(* Logix 5000 project; controller FRC_CC_2020 vendor 1 type 14 code 150 rev 31.11; software revision 31.01; part 4 of 4 *)
(* tags used below, declared in another part *)
   Conn_Open : BOOL[32];
   Next_Write : BOOL[32];
   ONS : BOOL[64];
   ONS_B : BOOL[32];
   ONS_ERR : BOOL[32];
   RW_Instance : INT[20];
   RW_Select : DINT;
   MBTI_Read_Data_MSG_07 : MESSAGE;
   MBTI_Read_Data_MSG_08 : MESSAGE;
   MBTI_Read_Data_MSG_09 : MESSAGE;
   MBTI_Read_Done : BOOL[32];
   MBTI_Read_Resp : READ_RESP_STR[10];
   MBTI_Write_Data_MSG_06 : MESSAGE;
   MBTI_Write_Data_MSG_07 : MESSAGE;
   MBTI_Write_Data_MSG_08 : MESSAGE;
   MBTI_Write_Data_MSG_09 : MESSAGE;
   MBTI_Write_Data_Out : WRT_DATA[10];
(* ModbusSlaveTCP, continued *)

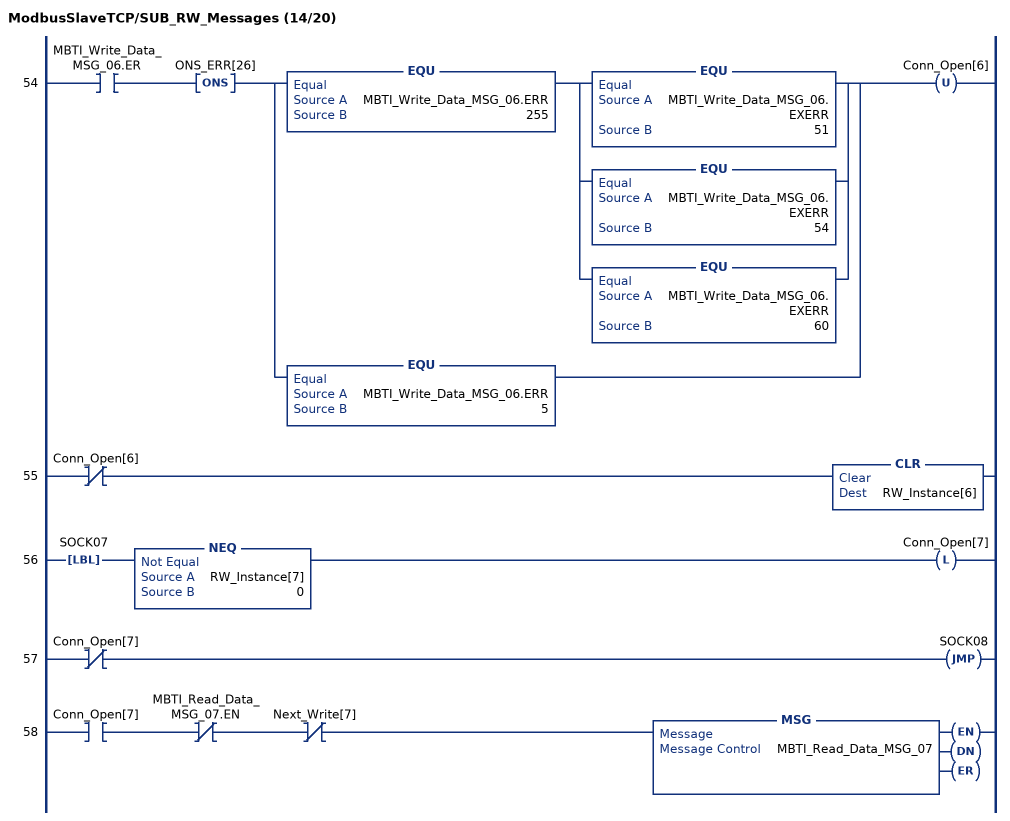
   [picture p61: ModbusSlaveTCP/SUB_RW_Messages rungs 54-58]
   54: XIC(MBTI_Write_Data_MSG_06.ER)ONS(ONS_ERR[26])[EQU(MBTI_Write_Data_MSG_06.ERR,255) [EQU(MBTI_Write_Data_MSG_06.EXERR,51) ,EQU(MBTI_Write_Data_MSG_06.EXERR,54) ,EQU(MBTI_Write_Data_MSG_06.EXERR,60) ] ,EQU(MBTI_Write_Data_MSG_06.ERR,5) ]OTU(Conn_Open[6]);
   55: XIO(Conn_Open[6])CLR(RW_Instance[6]);
   56: LBL(SOCK07)NEQ(RW_Instance[7],0)OTL(Conn_Open[7]);
   57: XIO(Conn_Open[7])JMP(SOCK08);
   58: XIC(Conn_Open[7])XIO(MBTI_Read_Data_MSG_07.EN)XIO(Next_Write[7])MSG(MBTI_Read_Data_MSG_07);
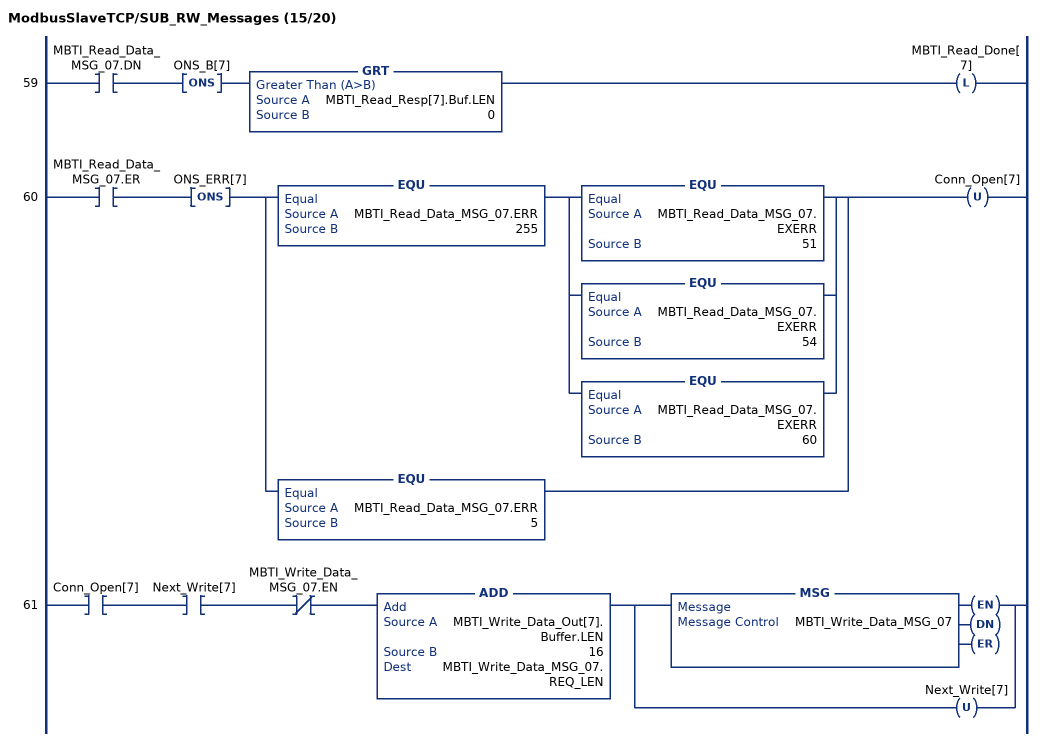
   59: XIC(MBTI_Read_Data_MSG_07.DN)ONS(ONS_B[7])GRT(MBTI_Read_Resp[7].Buf.LEN,0)OTL(MBTI_Read_Done[7]);
   60: XIC(MBTI_Read_Data_MSG_07.ER)ONS(ONS_ERR[7])[EQU(MBTI_Read_Data_MSG_07.ERR,255) [EQU(MBTI_Read_Data_MSG_07.EXERR,51) ,EQU(MBTI_Read_Data_MSG_07.EXERR,54) ,EQU(MBTI_Read_Data_MSG_07.EXERR,60) ] ,EQU(MBTI_Read_Data_MSG_07.ERR,5) ]OTU(Conn_Open[7]);
   61: XIC(Conn_Open[7])XIC(Next_Write[7])XIO(MBTI_Write_Data_MSG_07.EN)ADD(MBTI_Write_Data_Out[7].Buffer.LEN,16,MBTI_Write_Data_MSG_07.REQ_LEN)[MSG(MBTI_Write_Data_MSG_07) ,OTU(Next_Write[7]) ];
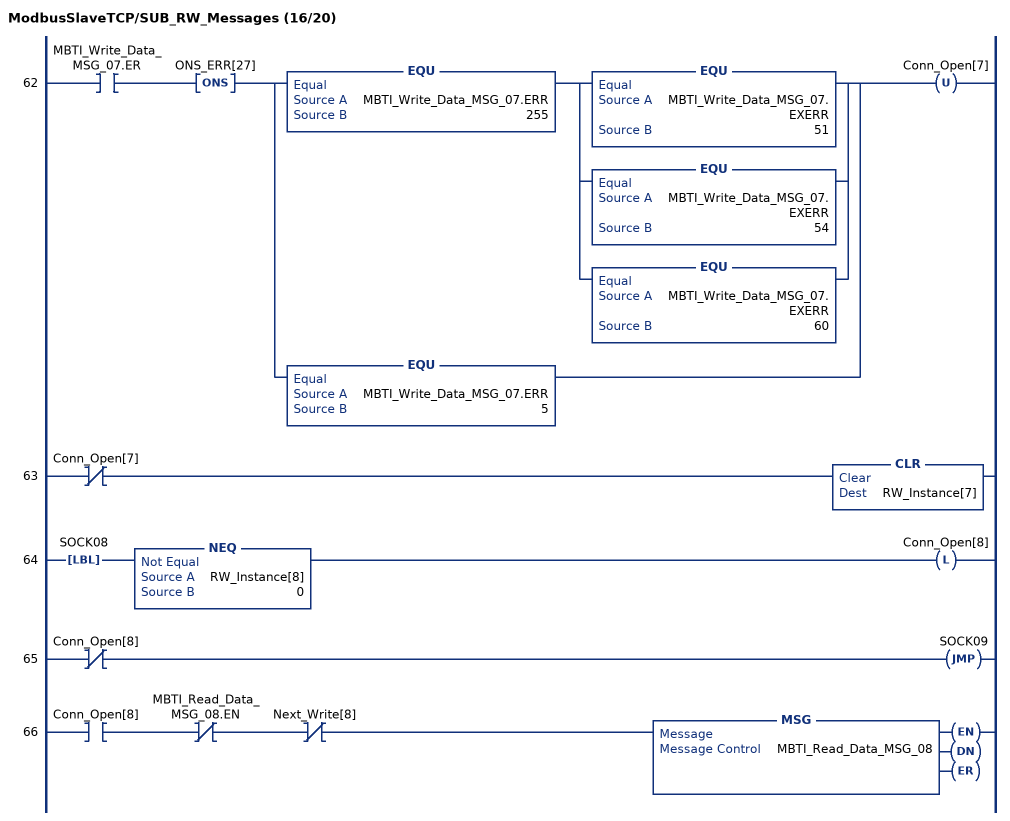
   62: XIC(MBTI_Write_Data_MSG_07.ER)ONS(ONS_ERR[27])[EQU(MBTI_Write_Data_MSG_07.ERR,255) [EQU(MBTI_Write_Data_MSG_07.EXERR,51) ,EQU(MBTI_Write_Data_MSG_07.EXERR,54) ,EQU(MBTI_Write_Data_MSG_07.EXERR,60) ] ,EQU(MBTI_Write_Data_MSG_07.ERR,5) ]OTU(Conn_Open[7]);
   63: XIO(Conn_Open[7])CLR(RW_Instance[7]);
   64: LBL(SOCK08)NEQ(RW_Instance[8],0)OTL(Conn_Open[8]);
   65: XIO(Conn_Open[8])JMP(SOCK09);
   66: XIC(Conn_Open[8])XIO(MBTI_Read_Data_MSG_08.EN)XIO(Next_Write[8])MSG(MBTI_Read_Data_MSG_08);
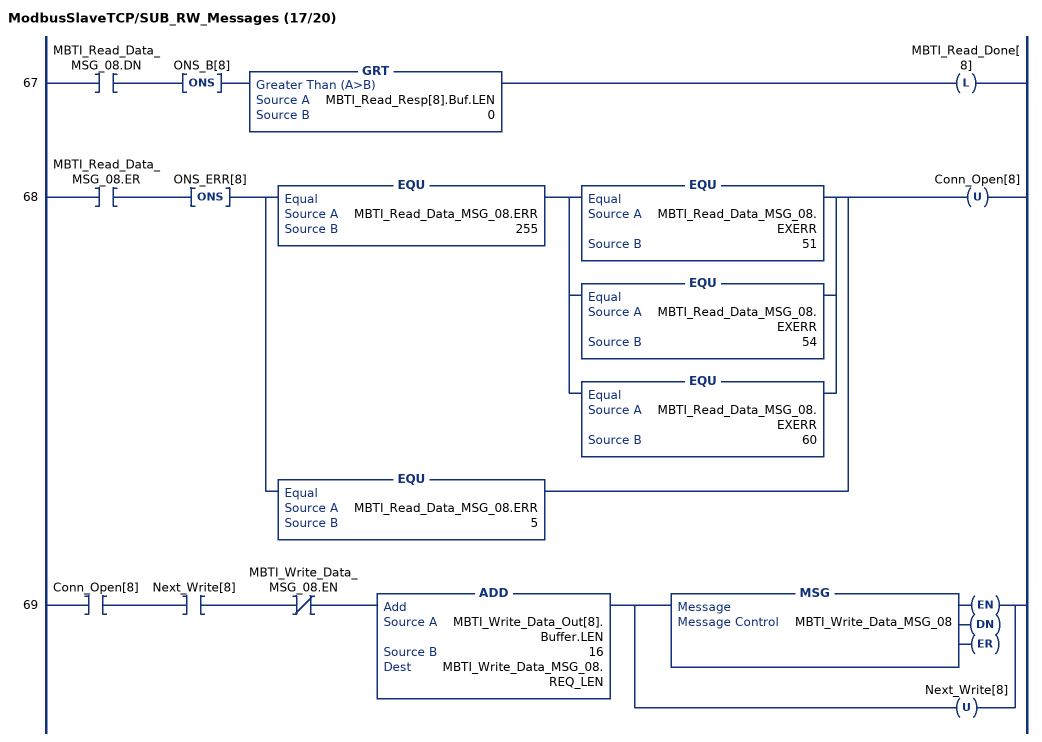
   67: XIC(MBTI_Read_Data_MSG_08.DN)ONS(ONS_B[8])GRT(MBTI_Read_Resp[8].Buf.LEN,0)OTL(MBTI_Read_Done[8]);
   68: XIC(MBTI_Read_Data_MSG_08.ER)ONS(ONS_ERR[8])[EQU(MBTI_Read_Data_MSG_08.ERR,255) [EQU(MBTI_Read_Data_MSG_08.EXERR,51) ,EQU(MBTI_Read_Data_MSG_08.EXERR,54) ,EQU(MBTI_Read_Data_MSG_08.EXERR,60) ] ,EQU(MBTI_Read_Data_MSG_08.ERR,5) ]OTU(Conn_Open[8]);
   69: XIC(Conn_Open[8])XIC(Next_Write[8])XIO(MBTI_Write_Data_MSG_08.EN)ADD(MBTI_Write_Data_Out[8].Buffer.LEN,16,MBTI_Write_Data_MSG_08.REQ_LEN)[MSG(MBTI_Write_Data_MSG_08) ,OTU(Next_Write[8]) ];
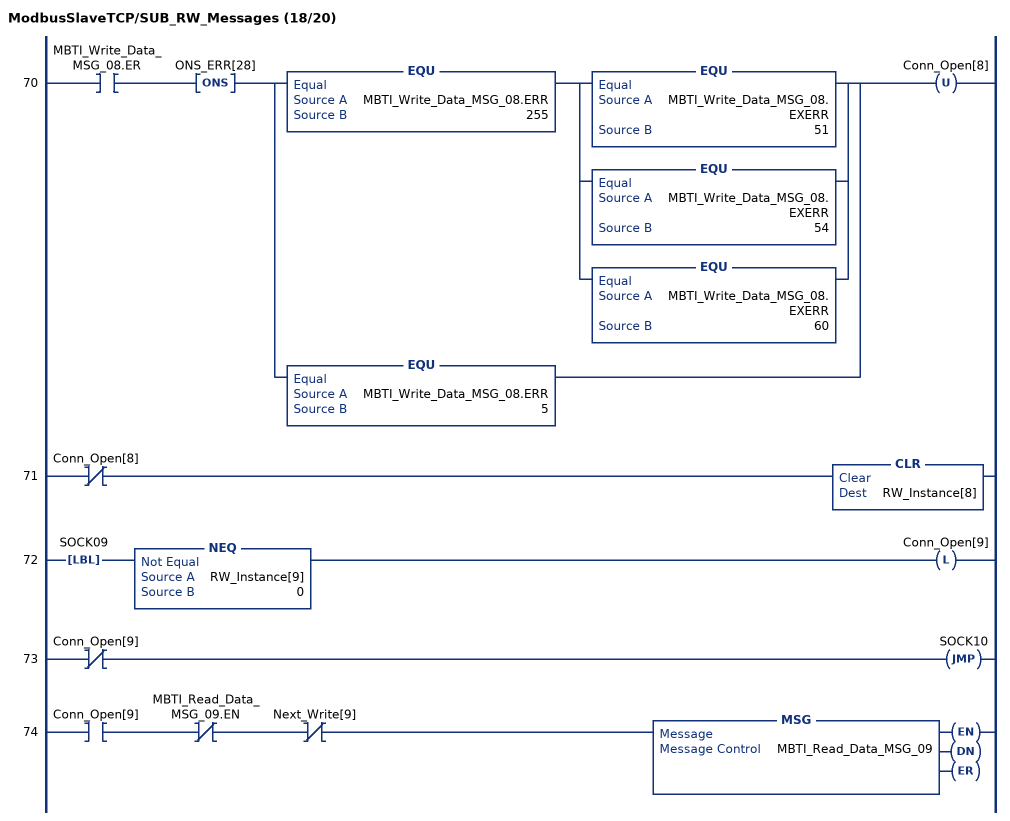
   70: XIC(MBTI_Write_Data_MSG_08.ER)ONS(ONS_ERR[28])[EQU(MBTI_Write_Data_MSG_08.ERR,255) [EQU(MBTI_Write_Data_MSG_08.EXERR,51) ,EQU(MBTI_Write_Data_MSG_08.EXERR,54) ,EQU(MBTI_Write_Data_MSG_08.EXERR,60) ] ,EQU(MBTI_Write_Data_MSG_08.ERR,5) ]OTU(Conn_Open[8]);
   71: XIO(Conn_Open[8])CLR(RW_Instance[8]);
   72: LBL(SOCK09)NEQ(RW_Instance[9],0)OTL(Conn_Open[9]);
   73: XIO(Conn_Open[9])JMP(SOCK10);
   74: XIC(Conn_Open[9])XIO(MBTI_Read_Data_MSG_09.EN)XIO(Next_Write[9])MSG(MBTI_Read_Data_MSG_09);
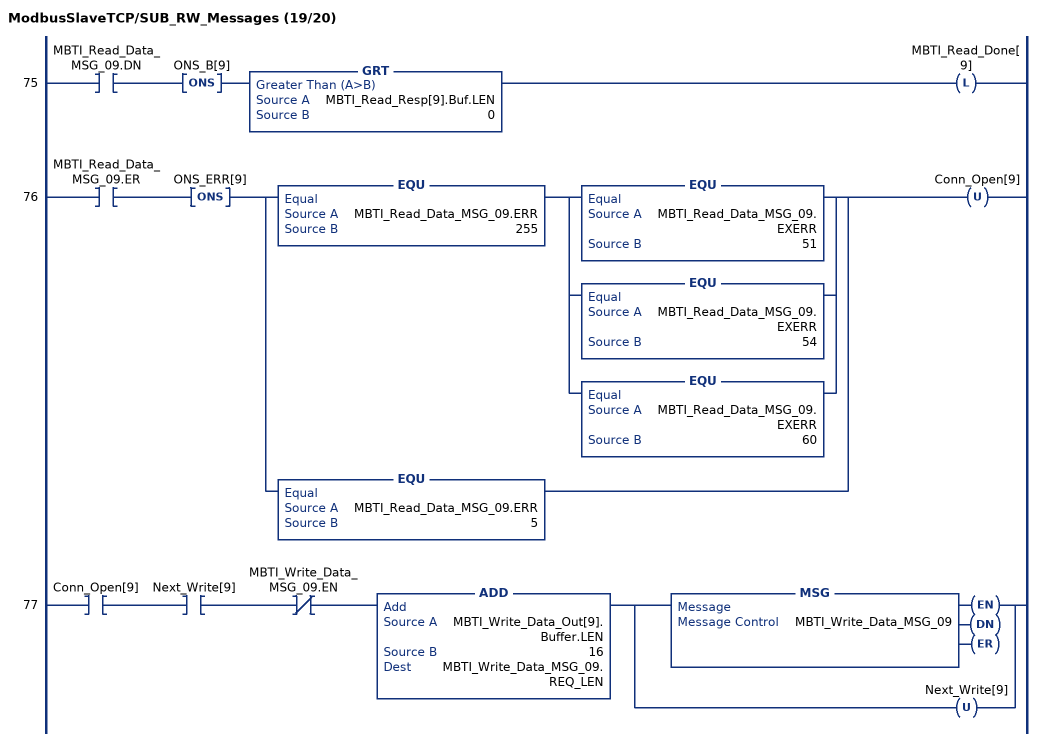
   75: XIC(MBTI_Read_Data_MSG_09.DN)ONS(ONS_B[9])GRT(MBTI_Read_Resp[9].Buf.LEN,0)OTL(MBTI_Read_Done[9]);
   76: XIC(MBTI_Read_Data_MSG_09.ER)ONS(ONS_ERR[9])[EQU(MBTI_Read_Data_MSG_09.ERR,255) [EQU(MBTI_Read_Data_MSG_09.EXERR,51) ,EQU(MBTI_Read_Data_MSG_09.EXERR,54) ,EQU(MBTI_Read_Data_MSG_09.EXERR,60) ] ,EQU(MBTI_Read_Data_MSG_09.ERR,5) ]OTU(Conn_Open[9]);
   77: XIC(Conn_Open[9])XIC(Next_Write[9])XIO(MBTI_Write_Data_MSG_09.EN)ADD(MBTI_Write_Data_Out[9].Buffer.LEN,16,MBTI_Write_Data_MSG_09.REQ_LEN)[MSG(MBTI_Write_Data_MSG_09) ,OTU(Next_Write[9]) ];
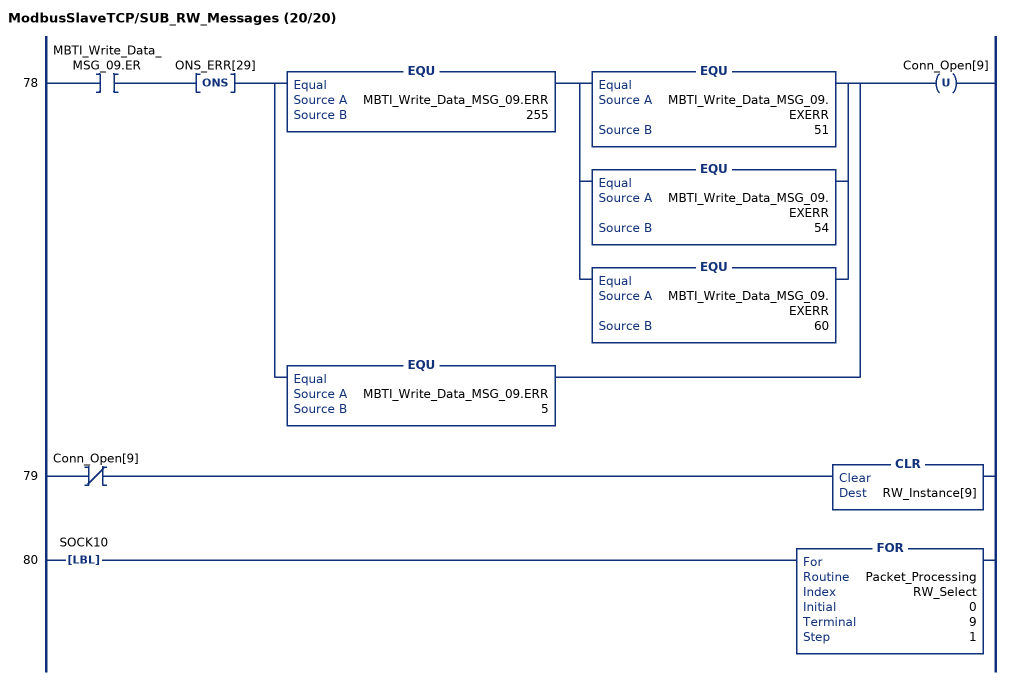
   78: XIC(MBTI_Write_Data_MSG_09.ER)ONS(ONS_ERR[29])[EQU(MBTI_Write_Data_MSG_09.ERR,255) [EQU(MBTI_Write_Data_MSG_09.EXERR,51) ,EQU(MBTI_Write_Data_MSG_09.EXERR,54) ,EQU(MBTI_Write_Data_MSG_09.EXERR,60) ] ,EQU(MBTI_Write_Data_MSG_09.ERR,5) ]OTU(Conn_Open[9]);
   79: XIO(Conn_Open[9])CLR(RW_Instance[9]);
   80: LBL(SOCK10)FOR(Packet_Processing,RW_Select,0,9,1);
END_ROUTINE
END_PROGRAM
